FUNCTION_BLOCK itfRampImplement IMPLEMENTS itfRamp
VAR_INPUT
END_VAR
VAR_OUTPUT
END_VAR
VAR
	OutputValue : INT;
	RampDone : BOOL;
	RampRate : INT;
	TargetFreq : INT;
	PulsePeriod : INT;
	Timer : TON;
END_VAR

METHOD mDoneTargetFreq : BOOL
IF pOutputValue >= pTargetFreq THEN
	pRampDone := TRUE;
	ELSE
		pRampDone := FALSE;
END_IF
END_METHOD

METHOD mRampDown : INT
mTimerScale();
mDoneTargetFreq();

IF TIMER.Q THEN
	IF pOutputValue > 0 THEN
pOutputValue := pOutputValue - 1;
	END_IF
END_IF
END_METHOD

METHOD mRampUp : INT
mTimerScale();
mDoneTargetFreq();

IF TIMER.Q THEN
	IF pOutputValue < pTargetFreq THEN
pOutputValue := pOutputValue + 1;
	END_IF
END_IF
END_METHOD

METHOD mTimerScale : INT
pPulsePeriod := (pRampRate * 1000) / TargetFreq;

TIMER(IN:= NOT TIMER.Q, PT:= INT_TO_TIME(pPulsePeriod));
END_METHOD

PROPERTY pOutputValue : INT
GET
pOutputValue := OutputValue;
END_GET
SET
OutputValue := pOutputValue;
END_SET
END_PROPERTY

PROPERTY pPulsePeriod : INT
GET
pPulsePeriod := PulsePeriod;
END_GET
SET
PulsePeriod := pPulsePeriod;
END_SET
END_PROPERTY

PROPERTY pRampDone : BOOL
GET
pRampDone := RampDone;
END_GET
SET
RampDone := pRampDone;
END_SET
END_PROPERTY

PROPERTY pRampRate : INT
GET
pRampRate := RampRate;
END_GET
SET
RampRate := pRampRate;
END_SET
END_PROPERTY

PROPERTY pTargetFreq : INT
GET
IF TargetFreq > 0 THEN
pTargetFreq := TargetFreq;
ELSE
	pTargetFreq := 1;
END_IF
END_GET
SET
VAR
	END_IFTargetFreq: INT;
END_VAR
IF pTargetFreq > 0 THEN
TargetFreq := pTargetFreq;
ELSE
	TargetFreq := 1;
END_IF
END_SET
END_PROPERTY

END_FUNCTION_BLOCK

(* stored: Version 1.1.0.1, ProductVersion 3.1.4024.12
   POU itfRampImplement: Id {595e310e-b0c8-4980-921f-214373609f3e}, SpecialFunc None
   Method mDoneTargetFreq: Id {81acbe68-1b98-4ba5-a8e6-58e4f7c79595}
   Method mRampDown: Id {cf4d1c2a-8557-44d9-a779-c89f9a9ffed8}
   Method mRampUp: Id {bbf02685-e48d-463f-9a3f-fbba743822b2}
   Method mTimerScale: Id {ea2a2985-6179-48b4-bb75-47f457a03ec5}
   Property pOutputValue: Id {96e85b45-f133-4a06-b7c3-5d2e77884a5e}
   Get Get: Id {a25bcb58-8011-4d25-9371-209fa84788f7}
   Set Set: Id {8c416970-e9e1-4044-812c-cc5a63db155d}
   Property pPulsePeriod: Id {f7552bfd-08e0-4f8e-ace6-d268ef126ce1}
   Get Get: Id {fcfd2e89-98e0-455f-8cd1-c536ab42e0d4}
   Set Set: Id {9bdebe48-0215-4c02-be41-98d60d173ed0}
   Property pRampDone: Id {cab89f5d-d190-4d69-8e64-5c87cac2d44a}
   Get Get: Id {94942c35-6010-48a8-a51a-b41667e52cad}
   Set Set: Id {b8f72e14-90bc-49fe-8ee0-27045e62f355}
   Property pRampRate: Id {2f5a2c69-d94c-4566-8b9f-331af3018a61}
   Get Get: Id {89dc5717-c7bb-4357-b1ae-4457a4f2d1f3}
   Set Set: Id {5282d2c2-5bdf-4bb3-8aab-6d5b15f040eb}
   Property pTargetFreq: Id {612859f9-8eef-4225-8ea4-2a74f9badd9a}
   Get Get: Id {103237b5-eb27-4653-b1f8-98e1d4337996}
   Set Set: Id {8d4b36d9-c5e2-479c-892a-d5adb74a1d3c} *)
